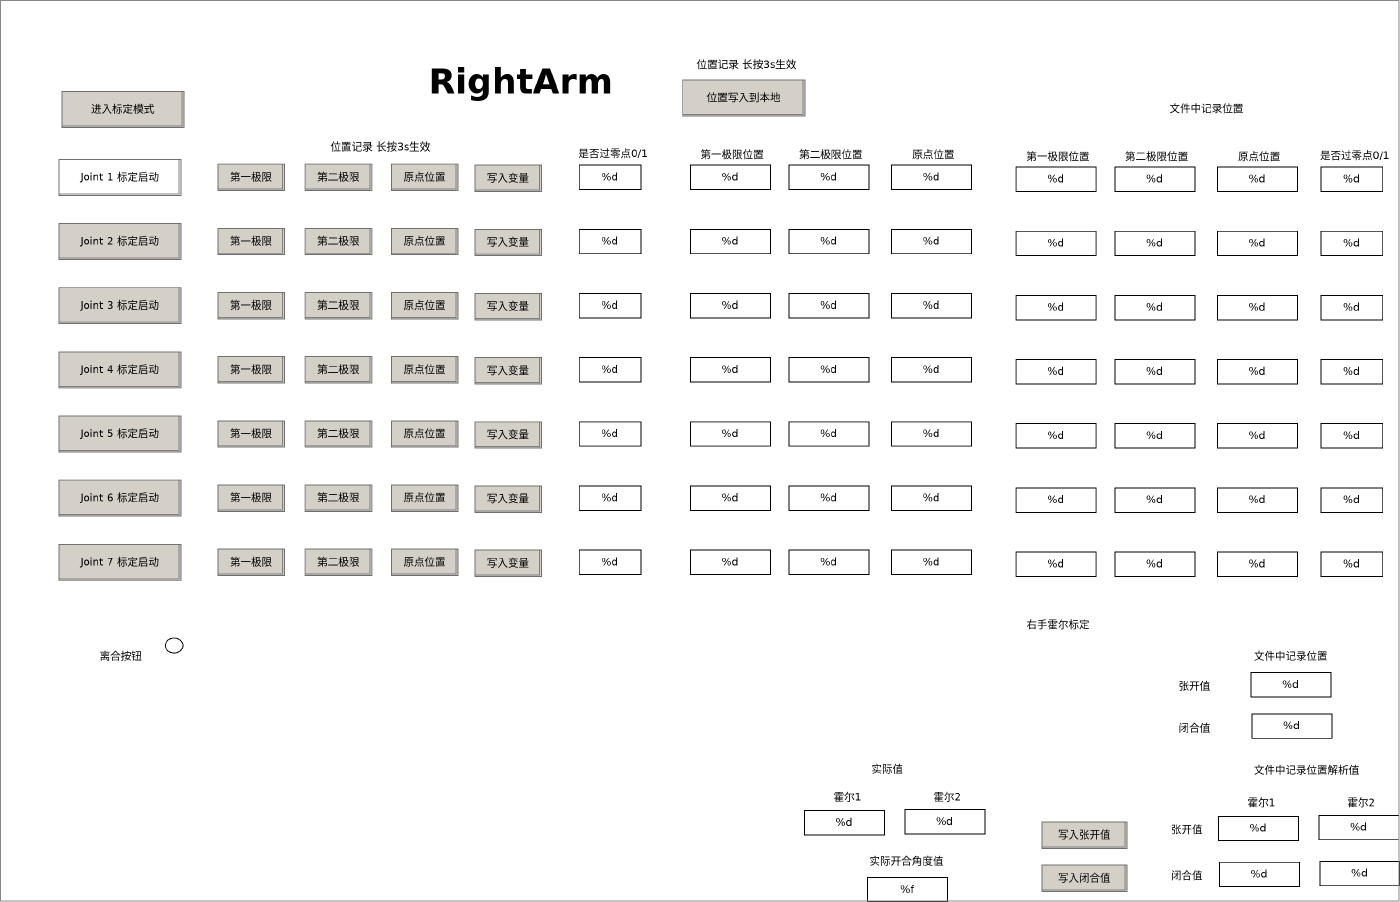
VISUALIZATION rightArmCail  // 1461x942
    Button (64,95 128x38), "进入标定模式", colour toggle: GVL_armCali.g_armEnterCaliMode[2]
        toggle GVL_armCali.g_armEnterCaliMode[2]
    Button (61,166 128x38), "Joint 1 标定启动", colour toggle: GVL_armCali.g_jointIntoCaliState[2][1]
        toggle GVL_armCali.g_jointIntoCaliState[2][1]
    Label (445,59 197x52), "RightArm"
    Button (61,233 128x38), "Joint 2 标定启动", colour toggle: GVL_armCali.g_jointIntoCaliState[2][2]
        toggle GVL_armCali.g_jointIntoCaliState[2][2]
    Button (227,171 70x28), "第一极限", colour toggle: GVL_armCali.g_linkEncFristCaliTrigger[2][1]
        tap GVL_armCali.g_linkEncFristPosCali[2][1]
    Button (318,171 70x28), "第二极限", colour toggle: GVL_armCali.g_linkEncSecondCaliTrigger[2][1]
        tap GVL_armCali.g_linkEncSecondPosCali[2][1]
    Rectangle (604,172 65x26), "%d", text variable: GVL_armCali.g_linkZeroCrossOrNot[2][1]
    Label (599,149 82x23), "是否过零点0/1"
    Rectangle (720,172 84x26), "%d", text variable: GVL_armCali.g_linkLimitFristPos[2][1]
    Label (723,150 82x23), "第一极限位置"
    Rectangle (823,172 84x26), "%d", text variable: GVL_armCali.g_linkLimitSecondPos[2][1]
    Label (826,150 82x23), "第二极限位置"
    Label (322,142 150x23), "位置记录 长按3s生效"
    Rectangle (930,172 84x26), "%d", text variable: GVL_armCali.g_linkHomePos[2][1]
    Label (933,150 82x23), "原点位置"
    Button (408,171 70x28), "原点位置", colour toggle: GVL_armCali.g_linkEncHomePosCaliTrigger[2][1]
        tap GVL_armCali.g_linkEncHomePosCali[2][1]
    Button (712,83 128x38), "位置写入到本地", colour toggle: GVL_armCali.g_caliDataWriteTrigger
        tap GVL_armCali.g_caliDataWrite
    Label (704,56 150x23), "位置记录 长按3s生效"
    Button (227,238 70x28), "第一极限", colour toggle: GVL_armCali.g_linkEncFristCaliTrigger[2][2]
        tap GVL_armCali.g_linkEncFristPosCali[2][2]
    Button (318,238 70x28), "第二极限", colour toggle: GVL_armCali.g_linkEncSecondCaliTrigger[2][2]
        tap GVL_armCali.g_linkEncSecondPosCali[2][2]
    Rectangle (604,239 65x26), "%d", text variable: GVL_armCali.g_linkZeroCrossOrNot[2][2]
    Rectangle (720,239 84x26), "%d", text variable: GVL_armCali.g_linkLimitFristPos[2][2]
    Rectangle (823,239 84x26), "%d", text variable: GVL_armCali.g_linkLimitSecondPos[2][2]
    Rectangle (930,239 84x26), "%d", text variable: GVL_armCali.g_linkHomePos[2][2]
    Button (408,238 70x28), "原点位置", colour toggle: GVL_armCali.g_linkEncHomePosCaliTrigger[2][2]
        tap GVL_armCali.g_linkEncHomePosCali[2][2]
    Button (61,300 128x38), "Joint 3 标定启动", colour toggle: GVL_armCali.g_jointIntoCaliState[2][3]
        toggle GVL_armCali.g_jointIntoCaliState[2][3]
    Button (227,305 70x28), "第一极限", colour toggle: GVL_armCali.g_linkEncFristCaliTrigger[2][3]
        tap GVL_armCali.g_linkEncFristPosCali[2][3]
    Button (318,305 70x28), "第二极限", colour toggle: GVL_armCali.g_linkEncSecondCaliTrigger[2][3]
        tap GVL_armCali.g_linkEncSecondPosCali[2][3]
    Rectangle (604,306 65x26), "%d", text variable: GVL_armCali.g_linkZeroCrossOrNot[2][3]
    Rectangle (720,306 84x26), "%d", text variable: GVL_armCali.g_linkLimitFristPos[2][3]
    Rectangle (823,306 84x26), "%d", text variable: GVL_armCali.g_linkLimitSecondPos[2][3]
    Rectangle (930,306 84x26), "%d", text variable: GVL_armCali.g_linkHomePos[2][3]
    Button (408,305 70x28), "原点位置", colour toggle: GVL_armCali.g_linkEncHomePosCaliTrigger[2][3]
        tap GVL_armCali.g_linkEncHomePosCali[2][3]
    Button (61,367 128x38), "Joint 4 标定启动", colour toggle: GVL_armCali.g_jointIntoCaliState[2][4]
        toggle GVL_armCali.g_jointIntoCaliState[2][4]
    Button (227,372 70x28), "第一极限", colour toggle: GVL_armCali.g_linkEncFristCaliTrigger[2][4]
        tap GVL_armCali.g_linkEncFristPosCali[2][4]
    Button (318,372 70x28), "第二极限", colour toggle: GVL_armCali.g_linkEncSecondCaliTrigger[2][4]
        tap GVL_armCali.g_linkEncSecondPosCali[2][4]
    Rectangle (604,373 65x26), "%d", text variable: GVL_armCali.g_linkZeroCrossOrNot[2][4]
    Rectangle (720,373 84x26), "%d", text variable: GVL_armCali.g_linkLimitFristPos[2][4]
    Rectangle (823,373 84x26), "%d", text variable: GVL_armCali.g_linkLimitSecondPos[2][4]
    Rectangle (930,373 84x26), "%d", text variable: GVL_armCali.g_linkHomePos[2][4]
    Button (408,372 70x28), "原点位置", colour toggle: GVL_armCali.g_linkEncHomePosCaliTrigger[2][4]
        tap GVL_armCali.g_linkEncHomePosCali[2][4]
    Button (61,434 128x38), "Joint 5 标定启动", colour toggle: GVL_armCali.g_jointIntoCaliState[2][5]
        toggle GVL_armCali.g_jointIntoCaliState[2][5]
    Button (227,439 70x28), "第一极限", colour toggle: GVL_armCali.g_linkEncFristCaliTrigger[2][5]
        tap GVL_armCali.g_linkEncFristPosCali[2][5]
    Button (318,439 70x28), "第二极限", colour toggle: GVL_armCali.g_linkEncSecondCaliTrigger[2][5]
        tap GVL_armCali.g_linkEncSecondPosCali[2][5]
    Rectangle (604,440 65x26), "%d", text variable: GVL_armCali.g_linkZeroCrossOrNot[2][5]
    Rectangle (720,440 84x26), "%d", text variable: GVL_armCali.g_linkLimitFristPos[2][5]
    Rectangle (823,440 84x26), "%d", text variable: GVL_armCali.g_linkLimitSecondPos[2][5]
    Rectangle (930,440 84x26), "%d", text variable: GVL_armCali.g_linkHomePos[2][5]
    Button (408,439 70x28), "原点位置", colour toggle: GVL_armCali.g_linkEncHomePosCaliTrigger[2][5]
        tap GVL_armCali.g_linkEncHomePosCali[2][5]
    Button (61,501 128x38), "Joint 6 标定启动", colour toggle: GVL_armCali.g_jointIntoCaliState[2][6]
        toggle GVL_armCali.g_jointIntoCaliState[2][6]
    Button (227,506 70x28), "第一极限", colour toggle: GVL_armCali.g_linkEncFristCaliTrigger[2][6]
        tap GVL_armCali.g_linkEncFristPosCali[2][6]
    Button (318,506 70x28), "第二极限", colour toggle: GVL_armCali.g_linkEncSecondCaliTrigger[2][6]
        tap GVL_armCali.g_linkEncSecondPosCali[2][6]
    Rectangle (604,507 65x26), "%d", text variable: GVL_armCali.g_linkZeroCrossOrNot[2][6]
    Rectangle (720,507 84x26), "%d", text variable: GVL_armCali.g_linkLimitFristPos[2][6]
    Rectangle (823,507 84x26), "%d", text variable: GVL_armCali.g_linkLimitSecondPos[2][6]
    Rectangle (930,507 84x26), "%d", text variable: GVL_armCali.g_linkHomePos[2][6]
    Button (408,506 70x28), "原点位置", colour toggle: GVL_armCali.g_linkEncHomePosCaliTrigger[2][6]
        tap GVL_armCali.g_linkEncHomePosCali[2][6]
    Button (61,568 128x38), "Joint 7 标定启动", colour toggle: GVL_armCali.g_jointIntoCaliState[2][7]
        toggle GVL_armCali.g_jointIntoCaliState[2][7]
    Button (227,573 70x28), "第一极限", colour toggle: GVL_armCali.g_linkEncFristCaliTrigger[2][7]
        tap GVL_armCali.g_linkEncFristPosCali[2][7]
    Button (318,573 70x28), "第二极限", colour toggle: GVL_armCali.g_linkEncSecondCaliTrigger[2][7]
        tap GVL_armCali.g_linkEncSecondPosCali[2][7]
    Rectangle (604,574 65x26), "%d", text variable: GVL_armCali.g_linkZeroCrossOrNot[2][7]
    Rectangle (720,574 84x26), "%d", text variable: GVL_armCali.g_linkLimitFristPos[2][7]
    Rectangle (823,574 84x26), "%d", text variable: GVL_armCali.g_linkLimitSecondPos[2][7]
    Rectangle (930,574 84x26), "%d", text variable: GVL_armCali.g_linkHomePos[2][7]
    Button (408,573 70x28), "原点位置", colour toggle: GVL_armCali.g_linkEncHomePosCaliTrigger[2][7]
        tap GVL_armCali.g_linkEncHomePosCali[2][7]
    Rectangle (1060,174 84x26), "%d", text variable: GVL_ArmJointCaliData.g_minLinkEncoder[2,1]
    Label (1063,152 82x23), "第一极限位置"
    Rectangle (1163,174 84x26), "%d", text variable: GVL_ArmJointCaliData.g_maxLinkEncoder[2,1]
    Label (1166,152 82x23), "第二极限位置"
    Rectangle (1270,174 84x26), "%d", text variable: GVL_ArmJointCaliData.g_caliLinkEncoder[2,1]
    Label (1273,152 82x23), "原点位置"
    Rectangle (1060,241 84x26), "%d", text variable: GVL_ArmJointCaliData.g_minLinkEncoder[2,2]
    Rectangle (1163,241 84x26), "%d", text variable: GVL_ArmJointCaliData.g_maxLinkEncoder[2,2]
    Rectangle (1270,241 84x26), "%d", text variable: GVL_ArmJointCaliData.g_caliLinkEncoder[2,2]
    Rectangle (1060,308 84x26), "%d", text variable: GVL_ArmJointCaliData.g_minLinkEncoder[2,3]
    Rectangle (1163,308 84x26), "%d", text variable: GVL_ArmJointCaliData.g_maxLinkEncoder[2,3]
    Rectangle (1270,308 84x26), "%d", text variable: GVL_ArmJointCaliData.g_caliLinkEncoder[2,3]
    Rectangle (1060,375 84x26), "%d", text variable: GVL_ArmJointCaliData.g_minLinkEncoder[2,4]
    Rectangle (1163,375 84x26), "%d", text variable: GVL_ArmJointCaliData.g_maxLinkEncoder[2,4]
    Rectangle (1270,375 84x26), "%d", text variable: GVL_ArmJointCaliData.g_caliLinkEncoder[2,4]
    Rectangle (1060,442 84x26), "%d", text variable: GVL_ArmJointCaliData.g_minLinkEncoder[2,5]
    Rectangle (1163,442 84x26), "%d", text variable: GVL_ArmJointCaliData.g_maxLinkEncoder[2,5]
    Rectangle (1270,442 84x26), "%d", text variable: GVL_ArmJointCaliData.g_caliLinkEncoder[2,5]
    Rectangle (1060,509 84x26), "%d", text variable: GVL_ArmJointCaliData.g_minLinkEncoder[2,6]
    Rectangle (1163,509 84x26), "%d", text variable: GVL_ArmJointCaliData.g_maxLinkEncoder[2,6]
    Rectangle (1270,509 84x26), "%d", text variable: GVL_ArmJointCaliData.g_caliLinkEncoder[2,6]
    Rectangle (1060,576 84x26), "%d", text variable: GVL_ArmJointCaliData.g_minLinkEncoder[2,7]
    Rectangle (1163,576 84x26), "%d", text variable: GVL_ArmJointCaliData.g_maxLinkEncoder[2,7]
    Rectangle (1270,576 84x26), "%d", text variable: GVL_ArmJointCaliData.g_caliLinkEncoder[2,7]
    Label (1184,102 150x23), "文件中记录位置"
    Rectangle (1378,174 65x26), "%d", text variable: GVL_ArmJointCaliData.g_linkEncZeroCross[2,1]
    Label (1373,151 82x23), "是否过零点0/1"
    Rectangle (1378,241 65x26), "%d", text variable: GVL_ArmJointCaliData.g_linkEncZeroCross[2,2]
    Rectangle (1378,308 65x26), "%d", text variable: GVL_ArmJointCaliData.g_linkEncZeroCross[2,3]
    Rectangle (1378,375 65x26), "%d", text variable: GVL_ArmJointCaliData.g_linkEncZeroCross[2,4]
    Rectangle (1378,442 65x26), "%d", text variable: GVL_ArmJointCaliData.g_linkEncZeroCross[2,5]
    Rectangle (1378,509 65x26), "%d", text variable: GVL_ArmJointCaliData.g_linkEncZeroCross[2,6]
    Rectangle (1378,576 65x26), "%d", text variable: GVL_ArmJointCaliData.g_linkEncZeroCross[2,7]
    Button (495,172 70x28), "写入变量", colour toggle: GVL_armCali.g_linkPosWriteCaliDataTrigger[2][1]
        tap GVL_armCali.g_linkPosWriteCaliData[2][1]
    Button (495,239 70x28), "写入变量", colour toggle: GVL_armCali.g_linkPosWriteCaliDataTrigger[2][2]
        tap GVL_armCali.g_linkPosWriteCaliData[2][2]
    Button (495,306 70x28), "写入变量", colour toggle: GVL_armCali.g_linkPosWriteCaliDataTrigger[2][3]
        tap GVL_armCali.g_linkPosWriteCaliData[2][3]
    Button (495,373 70x28), "写入变量", colour toggle: GVL_armCali.g_linkPosWriteCaliDataTrigger[2][4]
        tap GVL_armCali.g_linkPosWriteCaliData[2][4]
    Button (495,440 70x28), "写入变量", colour toggle: GVL_armCali.g_linkPosWriteCaliDataTrigger[2][5]
        tap GVL_armCali.g_linkPosWriteCaliData[2][5]
    Button (495,507 70x28), "写入变量", colour toggle: GVL_armCali.g_linkPosWriteCaliDataTrigger[2][6]
        tap GVL_armCali.g_linkPosWriteCaliData[2][6]
    Button (495,574 70x28), "写入变量", colour toggle: GVL_armCali.g_linkPosWriteCaliDataTrigger[2][7]
        tap GVL_armCali.g_linkPosWriteCaliData[2][7]
    Label (86,674 80x23), "离合按钮"
    Ellipse (172,666 19x16), colour toggle: GVL_IO.g_clutchSingle[2]
    Rectangle (1271,852 84x26), "%d", text variable: GVL_armCali.g_minArmHallCaliAnalysis[2][1]
    Rectangle (1376,851 84x26), "%d", text variable: GVL_armCali.g_minArmHallCaliAnalysis[2][2]
    Label (1064,641 80x23), "右手霍尔标定"
    Label (1291,827 51x23), "霍尔1"
    Label (1395,827 51x23), "霍尔2"
    Rectangle (1272,900 84x26), "%d", text variable: GVL_armCali.g_maxArmHallCaliAnalysis[2][1]
    Rectangle (1377,899 84x26), "%d", text variable: GVL_armCali.g_maxArmHallCaliAnalysis[2][2]
    Label (1213,855 51x23), "张开值"
    Label (1213,903 51x23), "闭合值"
    Label (872,792 108x23), "实际值"
    Rectangle (839,846 84x26), "%d", text variable: MasterArmControl.m_masterRobot.m_masterArms[2].m_gripAngleCalc.m_gripHighHallSenorValue
    Rectangle (944,845 84x26), "%d", text variable: MasterArmControl.m_masterRobot.m_masterArms[2].m_gripAngleCalc.m_gripLowHallSenorValue
    Label (859,821 51x23), "霍尔1"
    Label (963,821 51x23), "霍尔2"
    Rectangle (905,916 84x26), "%f", text variable: MasterArmControl.m_masterRobot.m_masterArms[2].m_gripAngle
    Label (892,888 108x23), "实际开合角度值"
    Button (1087,858 89x28), "写入张开值", colour toggle: GVL_armCali.g_masterArmHallCaliTrigger[2][1]
        tap GVL_armCali.g_masterArmHallCali[2][1]
    Button (1087,903 89x28), "写入闭合值", colour toggle: GVL_armCali.g_masterArmHallCaliTrigger[2][2]
        tap GVL_armCali.g_masterArmHallCali[2][2]
    Label (1293,674 108x23), "文件中记录位置"
    Rectangle (1305,702 84x26), "%d", text variable: GVL_ArmJointCaliData.g_minHallSensorValue[2]
    Label (1221,705 51x23), "张开值"
    Label (1221,749 51x23), "闭合值"
    Rectangle (1306,745 84x26), "%d", text variable: GVL_ArmJointCaliData.g_maxHallSensorValue[2]
    Label (1299,793 129x23), "文件中记录位置解析值"
END_VISUALIZATION

(* stored: Version 1.1.0.1, ProductVersion 3.1.4024.11
   Visu rightArmCail: Id {58b436d8-3d98-4529-9a1e-cf6d70f6b95e} *)
